(* CoDeSys 2.3 export: READ_SD_CARD.EXP *)

(* POU Read_SD_Card, FBD *)
FUNCTION_BLOCK Read_SD_Card
VAR_INPUT
		enable				: BOOL				:= FALSE;					(* enable the FUNCTION block *)
		sFileName		: STRING			:= 'sdcard\plan.csv';		(* absolute path of file to operate on *)
END_VAR
VAR_OUTPUT
		done				: BOOL;
		error				: BOOL;
END_VAR
VAR_IN_OUT
		IncomingData		: STRING(STRING_SIZE_READ)	;			(* buffer for incoming read data*)
END_VAR
VAR
	Open_file: FILE_Open;
	FileMode			: FILE_MODE		:= FILE_MREAD;				(* open for r+w access, file stream pointer at end of the file *)

	Read_file			: FILE_Read;
	File_Handle		: CAA_HANDLE;

	xReadAbort		: BOOL;

	close_file: FILE_Close;
	count_closes: CTU;
	reset: BOOL;
	counter_value_close: DWORD;
	count_opened: CTU;
	counter_value_open: DWORD;
	zustand				: SR;

	error_open: BOOL;
	error_read: BOOL;
	error_close: BOOL;
	error_open_number: INT;
	error_read_number: INT;
	error_close_number: INT;
END_VAR
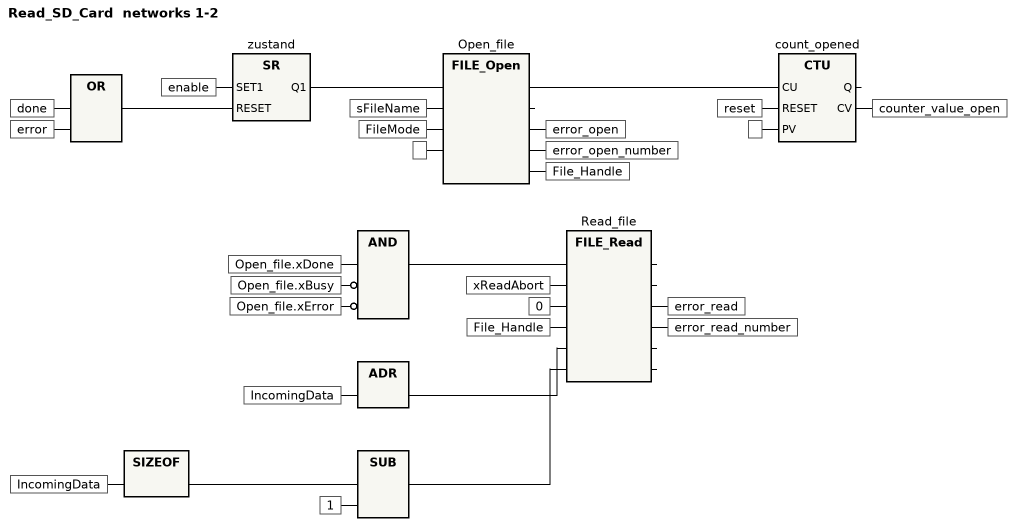
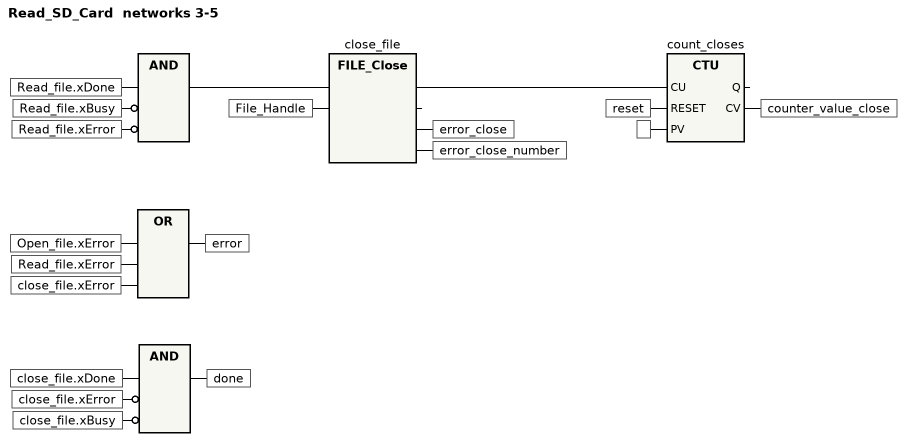
_FBD_ (* Function Block Diagram *)
NETWORK 1
	count_opened:CTU(CU: Open_file:FILE_Open(zustand:SR(SET1: enable, RESET: OR(done, error)), sFileName, FileMode, , out 3 => error_open, out 4 => error_open_number, out 5 => File_Handle), RESET: reset, PV: , CV => counter_value_open)
NETWORK 2
	Read_file:FILE_Read(AND(Open_file.xDone, NOT Open_file.xBusy, NOT Open_file.xError), xReadAbort, 0, File_Handle, ADR(IncomingData), SUB(SIZEOF(IncomingData), 1), out 3 => error_read, out 4 => error_read_number)
NETWORK 3
	count_closes:CTU(CU: close_file:FILE_Close(AND(Read_file.xDone, NOT Read_file.xBusy, NOT Read_file.xError), File_Handle, out 3 => error_close, out 4 => error_close_number), RESET: reset, PV: , CV => counter_value_close)
NETWORK 4
	OR(Open_file.xError, Read_file.xError, close_file.xError) => error
NETWORK 5
	AND(close_file.xDone, NOT close_file.xError, NOT close_file.xBusy) => done
_END_FBD_
(* the same logic as Structured Text *)
(* Network 1: see the listing above *)
(* Network 2: see the listing above *)
(* Network 3: see the listing above *)
(* Network 4 *)
error := Open_file.xError OR Read_file.xError OR close_file.xError;
(* Network 5 *)
done := close_file.xDone AND NOT close_file.xError AND NOT close_file.xBusy;
END_FUNCTION_BLOCK
